FUNCTION_BLOCK fb_BusTasterEvent
VAR_INPUT
	 I_sID         			:STRING(10);     // Geräte-ID (z.B. '12345')
	 I_sInstID				:STRING(2) 	:=	'17';
	 I_sReceivedString		:STRING(255);	
END_VAR
VAR_OUTPUT
	Q_bOut					:BOOL;
END_VAR
VAR
	findString0				:STRING ;
	findString1				:STRING ;
END_VAR


findString0 := CONCAT(I_sID,'.');
findString0 := CONCAT(findString0,'BTN');
findString0 := CONCAT(findString0,'.');
findString0 := CONCAT(findString0,I_sInstID);
findString0 := CONCAT(findString0,'.');
findString0 := CONCAT(findString0,'STATUS.0');

findString1 := CONCAT(I_sID,'.');
findString1 := CONCAT(findString1,'BTN');
findString1 := CONCAT(findString1,'.');
findString1 := CONCAT(findString1,I_sInstID);
findString1 := CONCAT(findString1,'.');
findString1 := CONCAT(findString1,'STATUS.1');

IF FIND(I_sReceivedString,findString0) >0 
THEN
	Q_bOut := FALSE;
ELSIF
	FIND(I_sReceivedString,findString1) >0 
THEN
	Q_bOut := TRUE;
END_IF

END_FUNCTION_BLOCK

(* stored: Version 1.1.0.1, ProductVersion 3.1.4024.12
   POU fb_BusTasterEvent: Id {c49e62e3-8862-4b59-ab27-a26658929b6b}, SpecialFunc None *)
